# EPICS substitutions: elioApp/Db/EL3164.substitutions
file EL3164.template { pattern
{ CHAN	}
{ 1	}
{ 2	}
{ 3	}
{ 4	}
}
